// TIA Portal V18 export
DATA_BLOCK "Main_Safety_RTG1_DB"   // DB1, F_DB
NAME : FUSI
VERSION : 0.1
// stored: AutoNumber true, DBAccessibleFromOPCUA true, InstanceOfName Main_Safety_RTG1, InstanceOfType FB
"Main_Safety_RTG1"
   // VAR
   //    ACK_GL_Instance : ACK_GL;
   //    FS_Room1_Instance : "FS_Room1";
   //    FS_Room2_Instance : "FS_Room2";
   //    FS_ACC_Instance : "FS_ACC";
   //    FS_VerticalBeam_Instance : "FS_VerticalBeam";
   // END_VAR
BEGIN
END_DATA_BLOCK
